Fanuc KAREL source: DAQ_STOP.kl

PROGRAM T
%NOLOCKGROUP
VAR
 v0 : INTEGER
 v1 : BOOLEAN
 v2 : INTEGER
BEGIN
 DAQ_STOP(v0, v1, v2)
END T
